Universal Robots PolyScope program: recibir_cadena_socket.urp

Program recibir_cadena_socket (installation=default directory=/programs/usbdisk createdIn=5.12.5.1101767 lastSavedIn=5.12.5.1101767 robotSerialNumber=20215500624)
Calibrated DH parameters: a=[0.000186, -0.025908, -0.392311, -0.000071, 0.00009, 0]; d=[0.162736, -361.104072, 360.092318, 1.145413, 0.099738, 0.099626]; alpha=[1.57079, -0.001175, 0.009075, 1.569386, -1.569463, 0]; deltaTheta=[0, 1.509811, 4.749978, 0.023394, 0, -0.000001]
BeforeStart
  conexion := False
  datos := [0,0,0,0]
  pos_pick := p[0,0,0,0,0,0]
Robot Program (runOnlyOnce=true)
  Loop While (checkContinuously=false) expression=conexion≟ False
    conexion := socket_open("192.168.1.249",50000)
    Wait Sleep waitTime=0.01
  str := "Listo"
  Script: socket_send_line(str)
  Loop While (checkContinuously=false) expression=datos[0]≠3
    datos := socket_read_ascii_float(3)
    Wait Sleep waitTime=0.5
  x := datos[1]
  y := datos[2]
  rz := datos[3]
  Script: socket_close()
  pos_pick := p[x,y,0,0,0,rz]
